// TIA Portal V18 export
FUNCTION "Conditon Check" : Void   // FC11, LAD
{ S7_Optimized_Access := 'TRUE' }
VERSION : 0.1
// stored: AutoNumber true, IsIECCheckEnabled false, SetENOAutomatically false, UDAEnableTagReadback false
   VAR_TEMP   // added for the SCL form of the ladder/FBD networks
      _w1 : Bool;
      _w2 : Bool;
      _w3 : Bool;
   END_VAR
BEGIN

REGION Network 1: Condition Check A without Valve
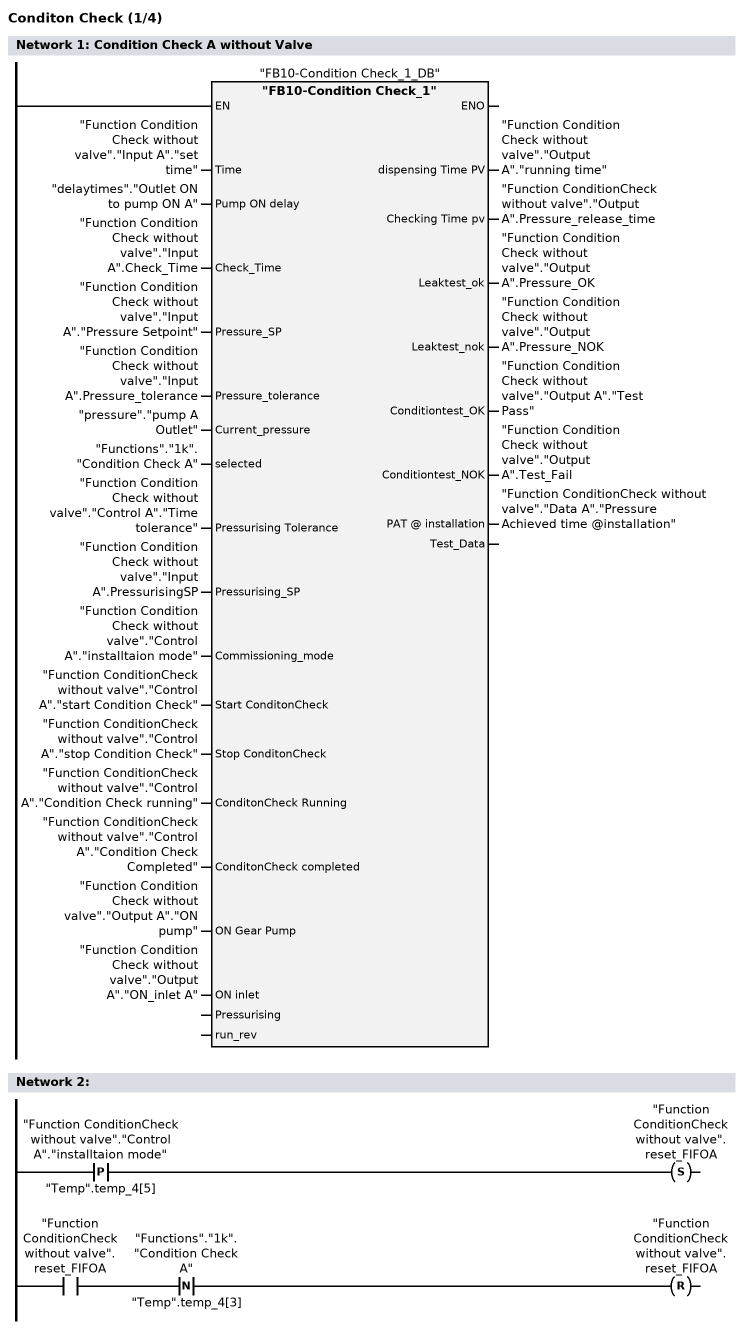
   RUNG wire#powerrail
      "FB10-Condition Check_1_DB"("Time" := "Function ConditionCheck without valve"."Input A"."set time", "Pump ON delay" := "delaytimes"."Outlet ON to pump ON A", Check_Time := "Function ConditionCheck without valve"."Input A".Check_Time, Pressure_SP := "Function ConditionCheck without valve"."Input A"."Pressure Setpoint", Pressure_tolerance := "Function ConditionCheck without valve"."Input A".Pressure_tolerance, Current_pressure := "pressure"."pump A Outlet", selected := "Functions"."1k"."Condition Check A", "Pressurising Tolerance" := "Function ConditionCheck without valve"."Control A"."Time tolerance", Pressurising_SP := "Function ConditionCheck without valve"."Input A".PressurisingSP, Commissioning_mode := "Function ConditionCheck without valve"."Control A"."installtaion mode", "Start ConditonCheck" := "Function ConditionCheck without valve"."Control A"."start Condition Check", "Stop ConditonCheck" := "Function ConditionCheck without valve"."Control A"."stop Condition Check", "ConditonCheck Running" := "Function ConditionCheck without valve"."Control A"."Condition Check running", "ConditonCheck completed" := "Function ConditionCheck without valve"."Control A"."Condition Check Completed", "ON Gear Pump" := "Function ConditionCheck without valve"."Output A"."ON pump", "ON inlet" := "Function ConditionCheck without valve"."Output A"."ON_inlet A", Pressurising :=, run_rev :=, "dispensing Time PV" => "Function ConditionCheck without valve"."Output A"."running time", "Checking Time pv" => "Function ConditionCheck without valve"."Output A".Pressure_release_time, Leaktest_ok => "Function ConditionCheck without valve"."Output A".Pressure_OK, Leaktest_nok => "Function ConditionCheck without valve"."Output A".Pressure_NOK, Conditiontest_OK => "Function ConditionCheck without valve"."Output A"."Test Pass", Conditiontest_NOK => "Function ConditionCheck without valve"."Output A".Test_Fail, "PAT @ installation" => "Function ConditionCheck without valve"."Data A"."Pressure Achieved time @installation", Test_Data =>)
   END_RUNG
   // the same network as SCL:
   "FB10-Condition Check_1_DB"("Time" := "Function ConditionCheck without valve"."Input A"."set time",   // "FB10-Condition Check_1"
                           "Pump ON delay" := "delaytimes"."Outlet ON to pump ON A",
                           Check_Time := "Function ConditionCheck without valve"."Input A".Check_Time,
                           Pressure_SP := "Function ConditionCheck without valve"."Input A"."Pressure Setpoint",
                           Pressure_tolerance := "Function ConditionCheck without valve"."Input A".Pressure_tolerance,
                           Current_pressure := "pressure"."pump A Outlet",
                           selected := "Functions"."1k"."Condition Check A",
                           "Pressurising Tolerance" := "Function ConditionCheck without valve"."Control A"."Time tolerance",
                           Pressurising_SP := "Function ConditionCheck without valve"."Input A".PressurisingSP,
                           Commissioning_mode := "Function ConditionCheck without valve"."Control A"."installtaion mode",
                           "Start ConditonCheck" := "Function ConditionCheck without valve"."Control A"."start Condition Check",
                           "Stop ConditonCheck" := "Function ConditionCheck without valve"."Control A"."stop Condition Check",
                           "ConditonCheck Running" := "Function ConditionCheck without valve"."Control A"."Condition Check running",
                           "ConditonCheck completed" := "Function ConditionCheck without valve"."Control A"."Condition Check Completed",
                           "ON Gear Pump" := "Function ConditionCheck without valve"."Output A"."ON pump",
                           "ON inlet" := "Function ConditionCheck without valve"."Output A"."ON_inlet A",
                           "dispensing Time PV" => "Function ConditionCheck without valve"."Output A"."running time",
                           "Checking Time pv" => "Function ConditionCheck without valve"."Output A".Pressure_release_time,
                           Leaktest_ok => "Function ConditionCheck without valve"."Output A".Pressure_OK,
                           Leaktest_nok => "Function ConditionCheck without valve"."Output A".Pressure_NOK,
                           Conditiontest_OK => "Function ConditionCheck without valve"."Output A"."Test Pass",
                           Conditiontest_NOK => "Function ConditionCheck without valve"."Output A".Test_Fail,
                           "PAT @ installation" => "Function ConditionCheck without valve"."Data A"."Pressure Achieved time @installation");
END_REGION

REGION Network 2
   RUNG wire#powerrail
      P_Contact(operand := "Function ConditionCheck without valve"."Control A"."installtaion mode", bit := "Temp".temp_4[5])
      S_Coil( "Function ConditionCheck without valve".reset_FIFOA )
   END_RUNG
   RUNG wire#powerrail
      Contact( "Function ConditionCheck without valve".reset_FIFOA )
      N_Contact(operand := "Functions"."1k"."Condition Check A", bit := "Temp".temp_4[3])
      R_Coil( "Function ConditionCheck without valve".reset_FIFOA )
   END_RUNG
   // the same network as SCL:
   #_w1 := "Function ConditionCheck without valve"."Control A"."installtaion mode" AND NOT "Temp".temp_4[5];   // rising edge of "Function ConditionCheck without valve"."Control A"."installtaion mode"
   "Temp".temp_4[5] := "Function ConditionCheck without valve"."Control A"."installtaion mode";
   IF #_w1 THEN "Function ConditionCheck without valve".reset_FIFOA := TRUE; END_IF;
   #_w2 := "Function ConditionCheck without valve".reset_FIFOA AND NOT "Functions"."1k"."Condition Check A" AND "Temp".temp_4[3];   // falling edge of "Functions"."1k"."Condition Check A"
   "Temp".temp_4[3] := "Functions"."1k"."Condition Check A";
   IF #_w2 THEN "Function ConditionCheck without valve".reset_FIFOA := FALSE; END_IF;
END_REGION

REGION Network 3
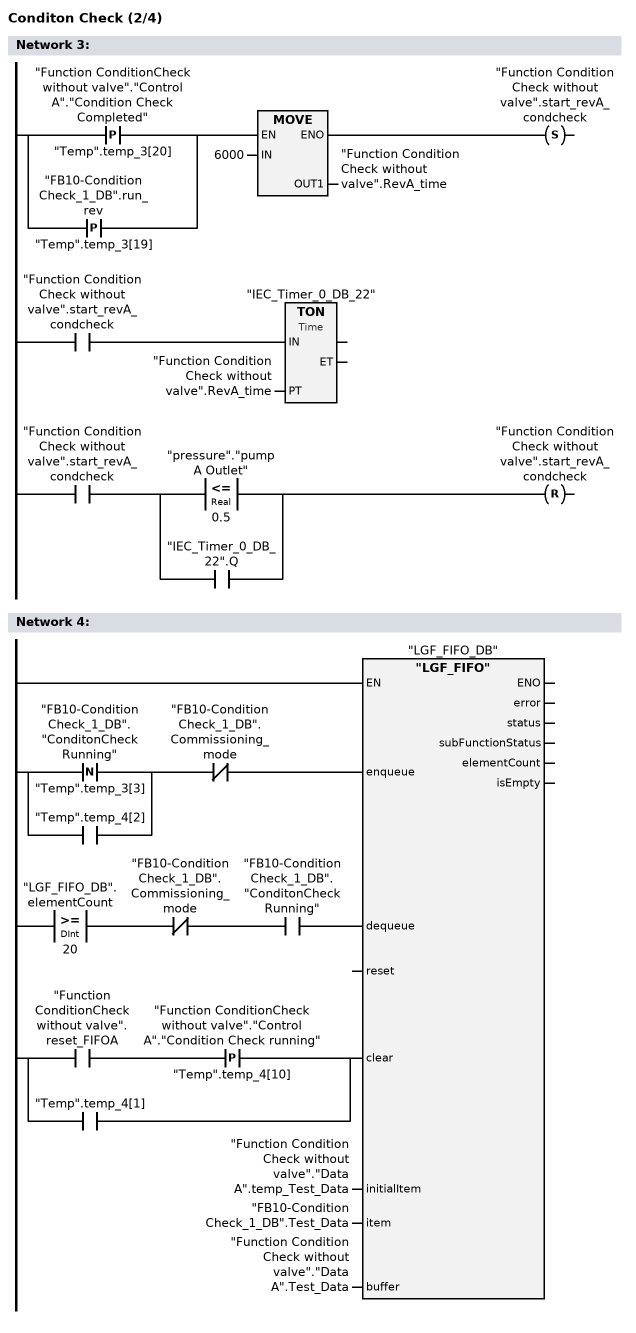
   RUNG wire#powerrail
      P_Contact(operand := "Function ConditionCheck without valve"."Control A"."Condition Check Completed", bit := "Temp".temp_3[20])
      wire#w1
      Move(in := 6000, out1 => "Function ConditionCheck without valve".RevA_time)
      S_Coil( "Function ConditionCheck without valve".start_revA_condcheck )
   END_RUNG
   RUNG wire#powerrail
      P_Contact(operand := "FB10-Condition Check_1_DB".run_rev, bit := "Temp".temp_3[19])
   END_RUNG wire#w1
   RUNG wire#powerrail
      Contact( "Function ConditionCheck without valve".start_revA_condcheck )
      { S7_Templates := "time_type := Time" } "IEC_Timer_0_DB_22".TON(pt := "Function ConditionCheck without valve".RevA_time, et =>)
   END_RUNG
   RUNG wire#powerrail
      Contact( "Function ConditionCheck without valve".start_revA_condcheck )
      wire#w2
      { S7_Templates := "SrcType := Real" } LE_Contact(in1 := "pressure"."pump A Outlet", in2 := 0.5)
      wire#w3
      R_Coil( "Function ConditionCheck without valve".start_revA_condcheck )
   END_RUNG
   RUNG wire#w2
      Contact( "IEC_Timer_0_DB_22".Q )
   END_RUNG wire#w3
   // the same network as SCL:
   #_w1 := "Function ConditionCheck without valve"."Control A"."Condition Check Completed" AND NOT "Temp".temp_3[20];   // rising edge of "Function ConditionCheck without valve"."Control A"."Condition Check Completed"
   "Temp".temp_3[20] := "Function ConditionCheck without valve"."Control A"."Condition Check Completed";
   #_w2 := "FB10-Condition Check_1_DB".run_rev AND NOT "Temp".temp_3[19];   // rising edge of "FB10-Condition Check_1_DB".run_rev
   "Temp".temp_3[19] := "FB10-Condition Check_1_DB".run_rev;
   IF #_w1 OR #_w2 THEN
       "Function ConditionCheck without valve".RevA_time := 6000;
       "Function ConditionCheck without valve".start_revA_condcheck := TRUE;
   END_IF;
   "IEC_Timer_0_DB_22".TON(IN := "Function ConditionCheck without valve".start_revA_condcheck,
                           PT := "Function ConditionCheck without valve".RevA_time);
   IF "Function ConditionCheck without valve".start_revA_condcheck AND (("pressure"."pump A Outlet" <= 0.5) OR "IEC_Timer_0_DB_22".Q) THEN
       "Function ConditionCheck without valve".start_revA_condcheck := FALSE;
   END_IF;
END_REGION

REGION Network 4
   RUNG wire#powerrail
      "LGF_FIFO_DB"(enqueue := wire#w2, dequeue := wire#w3, clear := wire#w4, reset :=, initialItem := "Function ConditionCheck without valve"."Data A".temp_Test_Data, item := "FB10-Condition Check_1_DB".Test_Data, buffer := "Function ConditionCheck without valve"."Data A".Test_Data, error =>, status =>, subFunctionStatus =>, elementCount =>, isEmpty =>)
   END_RUNG
   RUNG wire#powerrail
      N_Contact(operand := "FB10-Condition Check_1_DB"."ConditonCheck Running", bit := "Temp".temp_3[3])
      wire#w1
      I_Contact( "FB10-Condition Check_1_DB".Commissioning_mode )
   END_RUNG wire#w2
   RUNG wire#powerrail
      Contact( "Temp".temp_4[2] )
   END_RUNG wire#w1
   RUNG wire#powerrail
      { S7_Templates := "SrcType := DInt" } GE_Contact(in1 := "LGF_FIFO_DB".elementCount, in2 := 20)
      I_Contact( "FB10-Condition Check_1_DB".Commissioning_mode )
      Contact( "FB10-Condition Check_1_DB"."ConditonCheck Running" )
   END_RUNG wire#w3
   RUNG wire#powerrail
      Contact( "Function ConditionCheck without valve".reset_FIFOA )
      P_Contact(operand := "Function ConditionCheck without valve"."Control A"."Condition Check running", bit := "Temp".temp_4[10])
   END_RUNG wire#w4
   RUNG wire#powerrail
      Contact( "Temp".temp_4[1] )
   END_RUNG wire#w4
   // the same network as SCL:
   #_w1 := NOT "FB10-Condition Check_1_DB"."ConditonCheck Running" AND "Temp".temp_3[3];   // falling edge of "FB10-Condition Check_1_DB"."ConditonCheck Running"
   "Temp".temp_3[3] := "FB10-Condition Check_1_DB"."ConditonCheck Running";
   #_w3 := (#_w1 OR "Temp".temp_4[2]) AND NOT "FB10-Condition Check_1_DB".Commissioning_mode;
   #_w2 := "Function ConditionCheck without valve".reset_FIFOA AND "Function ConditionCheck without valve"."Control A"."Condition Check running" AND NOT "Temp".temp_4[10];   // rising edge of "Function ConditionCheck without valve"."Control A"."Condition Check running"
   "Temp".temp_4[10] := "Function ConditionCheck without valve"."Control A"."Condition Check running";
   "LGF_FIFO_DB"(enqueue := #_w3,   // "LGF_FIFO"
                 dequeue := ("LGF_FIFO_DB".elementCount >= 20) AND NOT "FB10-Condition Check_1_DB".Commissioning_mode AND "FB10-Condition Check_1_DB"."ConditonCheck Running",
                 clear := #_w2 OR "Temp".temp_4[1],
                 initialItem := "Function ConditionCheck without valve"."Data A".temp_Test_Data,
                 item := "FB10-Condition Check_1_DB".Test_Data,
                 buffer := "Function ConditionCheck without valve"."Data A".Test_Data);
END_REGION

REGION Network 5: Condition Check B without Valve
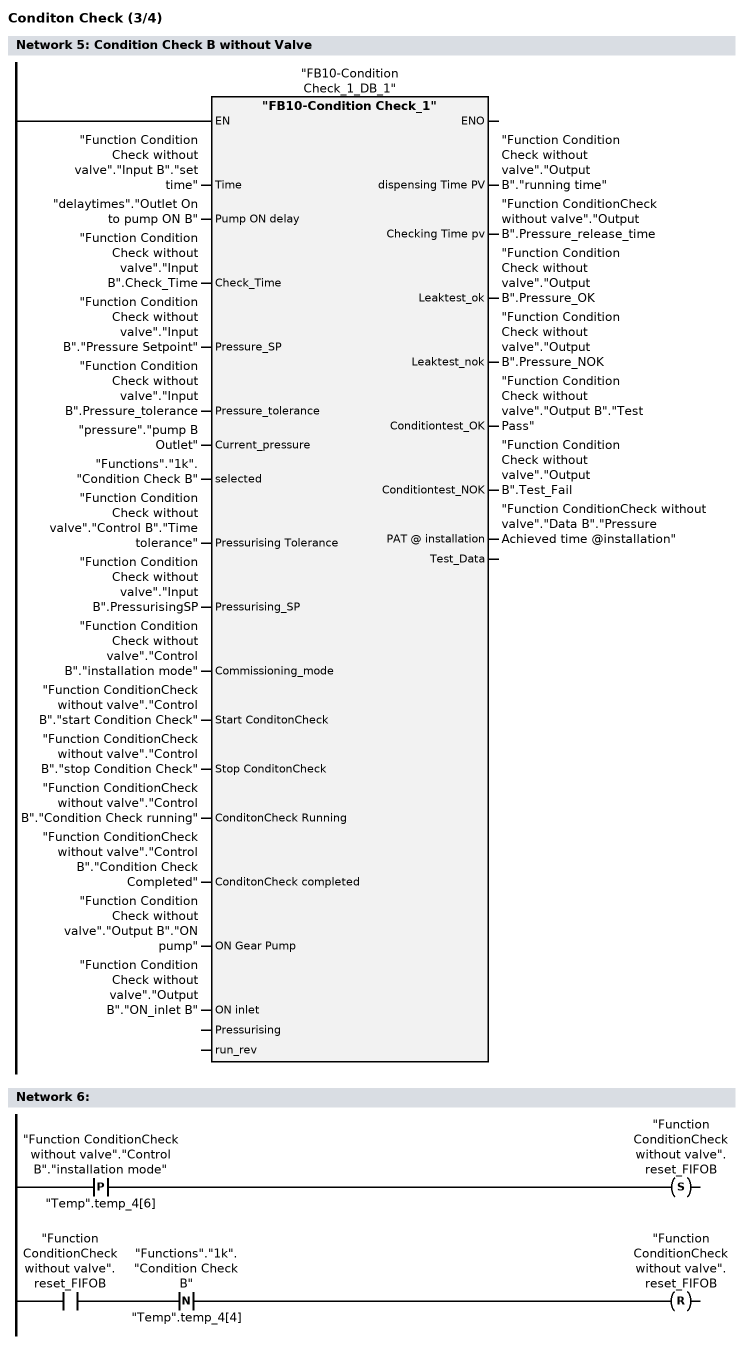
   RUNG wire#powerrail
      "FB10-Condition Check_1_DB_1"("Time" := "Function ConditionCheck without valve"."Input B"."set time", "Pump ON delay" := "delaytimes"."Outlet On to pump ON B", Check_Time := "Function ConditionCheck without valve"."Input B".Check_Time, Pressure_SP := "Function ConditionCheck without valve"."Input B"."Pressure Setpoint", Pressure_tolerance := "Function ConditionCheck without valve"."Input B".Pressure_tolerance, Current_pressure := "pressure"."pump B Outlet", selected := "Functions"."1k"."Condition Check B", "Pressurising Tolerance" := "Function ConditionCheck without valve"."Control B"."Time tolerance", Pressurising_SP := "Function ConditionCheck without valve"."Input B".PressurisingSP, Commissioning_mode := "Function ConditionCheck without valve"."Control B"."installation mode", "Start ConditonCheck" := "Function ConditionCheck without valve"."Control B"."start Condition Check", "Stop ConditonCheck" := "Function ConditionCheck without valve"."Control B"."stop Condition Check", "ConditonCheck Running" := "Function ConditionCheck without valve"."Control B"."Condition Check running", "ConditonCheck completed" := "Function ConditionCheck without valve"."Control B"."Condition Check Completed", "ON Gear Pump" := "Function ConditionCheck without valve"."Output B"."ON pump", "ON inlet" := "Function ConditionCheck without valve"."Output B"."ON_inlet B", Pressurising :=, run_rev :=, "dispensing Time PV" => "Function ConditionCheck without valve"."Output B"."running time", "Checking Time pv" => "Function ConditionCheck without valve"."Output B".Pressure_release_time, Leaktest_ok => "Function ConditionCheck without valve"."Output B".Pressure_OK, Leaktest_nok => "Function ConditionCheck without valve"."Output B".Pressure_NOK, Conditiontest_OK => "Function ConditionCheck without valve"."Output B"."Test Pass", Conditiontest_NOK => "Function ConditionCheck without valve"."Output B".Test_Fail, "PAT @ installation" => "Function ConditionCheck without valve"."Data B"."Pressure Achieved time @installation", Test_Data =>)
   END_RUNG
   // the same network as SCL:
   "FB10-Condition Check_1_DB_1"("Time" := "Function ConditionCheck without valve"."Input B"."set time",   // "FB10-Condition Check_1"
                           "Pump ON delay" := "delaytimes"."Outlet On to pump ON B",
                           Check_Time := "Function ConditionCheck without valve"."Input B".Check_Time,
                           Pressure_SP := "Function ConditionCheck without valve"."Input B"."Pressure Setpoint",
                           Pressure_tolerance := "Function ConditionCheck without valve"."Input B".Pressure_tolerance,
                           Current_pressure := "pressure"."pump B Outlet",
                           selected := "Functions"."1k"."Condition Check B",
                           "Pressurising Tolerance" := "Function ConditionCheck without valve"."Control B"."Time tolerance",
                           Pressurising_SP := "Function ConditionCheck without valve"."Input B".PressurisingSP,
                           Commissioning_mode := "Function ConditionCheck without valve"."Control B"."installation mode",
                           "Start ConditonCheck" := "Function ConditionCheck without valve"."Control B"."start Condition Check",
                           "Stop ConditonCheck" := "Function ConditionCheck without valve"."Control B"."stop Condition Check",
                           "ConditonCheck Running" := "Function ConditionCheck without valve"."Control B"."Condition Check running",
                           "ConditonCheck completed" := "Function ConditionCheck without valve"."Control B"."Condition Check Completed",
                           "ON Gear Pump" := "Function ConditionCheck without valve"."Output B"."ON pump",
                           "ON inlet" := "Function ConditionCheck without valve"."Output B"."ON_inlet B",
                           "dispensing Time PV" => "Function ConditionCheck without valve"."Output B"."running time",
                           "Checking Time pv" => "Function ConditionCheck without valve"."Output B".Pressure_release_time,
                           Leaktest_ok => "Function ConditionCheck without valve"."Output B".Pressure_OK,
                           Leaktest_nok => "Function ConditionCheck without valve"."Output B".Pressure_NOK,
                           Conditiontest_OK => "Function ConditionCheck without valve"."Output B"."Test Pass",
                           Conditiontest_NOK => "Function ConditionCheck without valve"."Output B".Test_Fail,
                           "PAT @ installation" => "Function ConditionCheck without valve"."Data B"."Pressure Achieved time @installation");
END_REGION

REGION Network 6
   RUNG wire#powerrail
      P_Contact(operand := "Function ConditionCheck without valve"."Control B"."installation mode", bit := "Temp".temp_4[6])
      S_Coil( "Function ConditionCheck without valve".reset_FIFOB )
   END_RUNG
   RUNG wire#powerrail
      Contact( "Function ConditionCheck without valve".reset_FIFOB )
      N_Contact(operand := "Functions"."1k"."Condition Check B", bit := "Temp".temp_4[4])
      R_Coil( "Function ConditionCheck without valve".reset_FIFOB )
   END_RUNG
   // the same network as SCL:
   #_w1 := "Function ConditionCheck without valve"."Control B"."installation mode" AND NOT "Temp".temp_4[6];   // rising edge of "Function ConditionCheck without valve"."Control B"."installation mode"
   "Temp".temp_4[6] := "Function ConditionCheck without valve"."Control B"."installation mode";
   IF #_w1 THEN "Function ConditionCheck without valve".reset_FIFOB := TRUE; END_IF;
   #_w2 := "Function ConditionCheck without valve".reset_FIFOB AND NOT "Functions"."1k"."Condition Check B" AND "Temp".temp_4[4];   // falling edge of "Functions"."1k"."Condition Check B"
   "Temp".temp_4[4] := "Functions"."1k"."Condition Check B";
   IF #_w2 THEN "Function ConditionCheck without valve".reset_FIFOB := FALSE; END_IF;
END_REGION

REGION Network 7
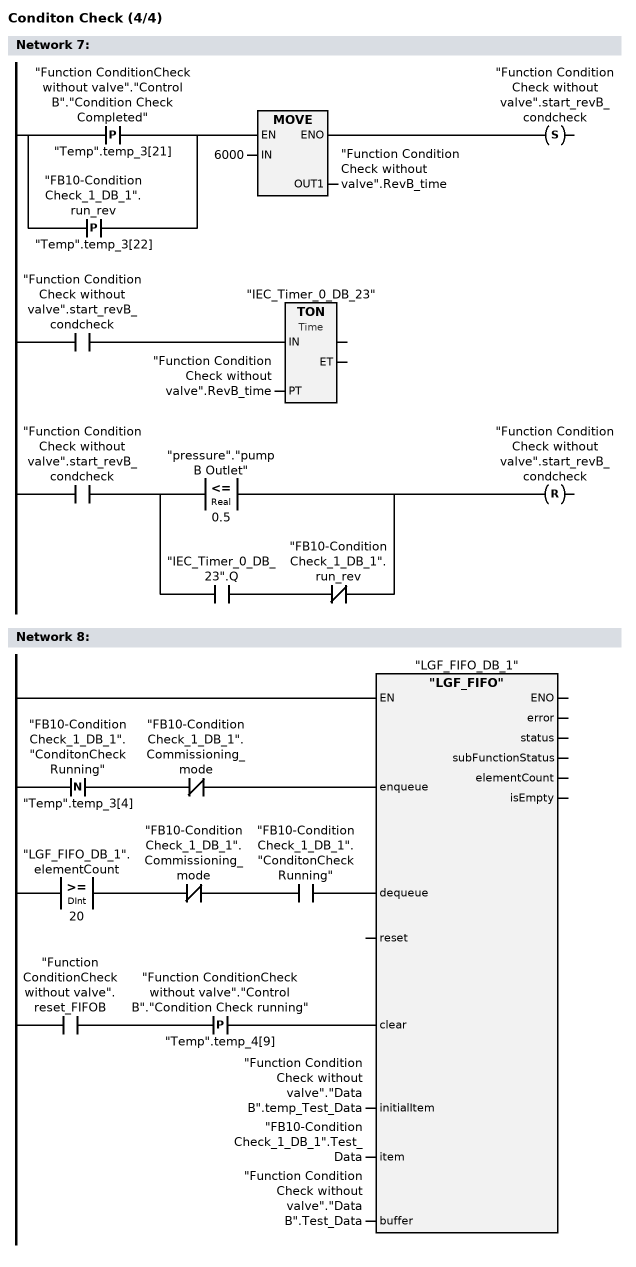
   RUNG wire#powerrail
      P_Contact(operand := "Function ConditionCheck without valve"."Control B"."Condition Check Completed", bit := "Temp".temp_3[21])
      wire#w1
      Move(in := 6000, out1 => "Function ConditionCheck without valve".RevB_time)
      S_Coil( "Function ConditionCheck without valve".start_revB_condcheck )
   END_RUNG
   RUNG wire#powerrail
      P_Contact(operand := "FB10-Condition Check_1_DB_1".run_rev, bit := "Temp".temp_3[22])
   END_RUNG wire#w1
   RUNG wire#powerrail
      Contact( "Function ConditionCheck without valve".start_revB_condcheck )
      { S7_Templates := "time_type := Time" } "IEC_Timer_0_DB_23".TON(pt := "Function ConditionCheck without valve".RevB_time, et =>)
   END_RUNG
   RUNG wire#powerrail
      Contact( "Function ConditionCheck without valve".start_revB_condcheck )
      wire#w2
      { S7_Templates := "SrcType := Real" } LE_Contact(in1 := "pressure"."pump B Outlet", in2 := 0.5)
      wire#w3
      R_Coil( "Function ConditionCheck without valve".start_revB_condcheck )
   END_RUNG
   RUNG wire#w2
      Contact( "IEC_Timer_0_DB_23".Q )
      I_Contact( "FB10-Condition Check_1_DB_1".run_rev )
   END_RUNG wire#w3
   // the same network as SCL:
   #_w1 := "Function ConditionCheck without valve"."Control B"."Condition Check Completed" AND NOT "Temp".temp_3[21];   // rising edge of "Function ConditionCheck without valve"."Control B"."Condition Check Completed"
   "Temp".temp_3[21] := "Function ConditionCheck without valve"."Control B"."Condition Check Completed";
   #_w2 := "FB10-Condition Check_1_DB_1".run_rev AND NOT "Temp".temp_3[22];   // rising edge of "FB10-Condition Check_1_DB_1".run_rev
   "Temp".temp_3[22] := "FB10-Condition Check_1_DB_1".run_rev;
   IF #_w1 OR #_w2 THEN
       "Function ConditionCheck without valve".RevB_time := 6000;
       "Function ConditionCheck without valve".start_revB_condcheck := TRUE;
   END_IF;
   "IEC_Timer_0_DB_23".TON(IN := "Function ConditionCheck without valve".start_revB_condcheck,
                           PT := "Function ConditionCheck without valve".RevB_time);
   IF "Function ConditionCheck without valve".start_revB_condcheck AND (("pressure"."pump B Outlet" <= 0.5) OR ("IEC_Timer_0_DB_23".Q AND NOT "FB10-Condition Check_1_DB_1".run_rev)) THEN
       "Function ConditionCheck without valve".start_revB_condcheck := FALSE;
   END_IF;
END_REGION

REGION Network 8
   RUNG wire#powerrail
      "LGF_FIFO_DB_1"(enqueue := wire#w1, dequeue := wire#w2, clear := wire#w3, reset :=, initialItem := "Function ConditionCheck without valve"."Data B".temp_Test_Data, item := "FB10-Condition Check_1_DB_1".Test_Data, buffer := "Function ConditionCheck without valve"."Data B".Test_Data, error =>, status =>, subFunctionStatus =>, elementCount =>, isEmpty =>)
   END_RUNG
   RUNG wire#powerrail
      N_Contact(operand := "FB10-Condition Check_1_DB_1"."ConditonCheck Running", bit := "Temp".temp_3[4])
      I_Contact( "FB10-Condition Check_1_DB_1".Commissioning_mode )
   END_RUNG wire#w1
   RUNG wire#powerrail
      { S7_Templates := "SrcType := DInt" } GE_Contact(in1 := "LGF_FIFO_DB_1".elementCount, in2 := 20)
      I_Contact( "FB10-Condition Check_1_DB_1".Commissioning_mode )
      Contact( "FB10-Condition Check_1_DB_1"."ConditonCheck Running" )
   END_RUNG wire#w2
   RUNG wire#powerrail
      Contact( "Function ConditionCheck without valve".reset_FIFOB )
      P_Contact(operand := "Function ConditionCheck without valve"."Control B"."Condition Check running", bit := "Temp".temp_4[9])
   END_RUNG wire#w3
   // the same network as SCL:
   #_w1 := NOT "FB10-Condition Check_1_DB_1"."ConditonCheck Running" AND "Temp".temp_3[4];   // falling edge of "FB10-Condition Check_1_DB_1"."ConditonCheck Running"
   "Temp".temp_3[4] := "FB10-Condition Check_1_DB_1"."ConditonCheck Running";
   #_w2 := "Function ConditionCheck without valve".reset_FIFOB AND "Function ConditionCheck without valve"."Control B"."Condition Check running" AND NOT "Temp".temp_4[9];   // rising edge of "Function ConditionCheck without valve"."Control B"."Condition Check running"
   "Temp".temp_4[9] := "Function ConditionCheck without valve"."Control B"."Condition Check running";
   "LGF_FIFO_DB_1"(enqueue := #_w1 AND NOT "FB10-Condition Check_1_DB_1".Commissioning_mode,   // "LGF_FIFO"
                   dequeue := ("LGF_FIFO_DB_1".elementCount >= 20) AND NOT "FB10-Condition Check_1_DB_1".Commissioning_mode AND "FB10-Condition Check_1_DB_1"."ConditonCheck Running",
                   clear := #_w2,
                   initialItem := "Function ConditionCheck without valve"."Data B".temp_Test_Data,
                   item := "FB10-Condition Check_1_DB_1".Test_Data,
                   buffer := "Function ConditionCheck without valve"."Data B".Test_Data);
END_REGION
END_FUNCTION
